{attribute addProperty BoxType "EL3423-0000-0020"}
{attribute addProperty Id "TxPDO_ToggleAT %I*BOOL8116Active_EnergyAT %I*REAL32417Apparent_EnergyAT %I*REAL32418Reactive_EnergyAT %I*REAL32419"}
{attribute addProperty CRC "3058033161"}
{attribute addProperty SizeInBites "104"}
{attribute addProperty SizeInBytes "13"}
TYPE Total_Interval_Energy_Reduced_B645E209 :
STRUCT
	{attribute addProperty Name "TxPDO_Toggle"}
	TxPDO_Toggle AT %I* : BOOL;
	{attribute addProperty Name "Active_Energy"}
	Active_Energy AT %I* : REAL;
	{attribute addProperty Name "Apparent_Energy"}
	Apparent_Energy AT %I* : REAL;
	{attribute addProperty Name "Reactive_Energy"}
	Reactive_Energy AT %I* : REAL;
END_STRUCT
END_TYPE

(* stored: Version 1.2.0.0, ProductVersion 3.1.4024.9
   DUT Total_Interval_Energy_Reduced_B645E209: Id {6f446987-f302-4620-a2e9-427335863763} *)
